Omron Sysmac Studio project ExamplePseudoUAMethod (Sysmac Studio 1.63.0.7, StandardProject)

# Controller Example: NX102-9000 version 1.64
Task PrimaryTask (priority 4, period or condition 4000): Methods, Math

VAR_GLOBAL
    Scalar_Static_Int32 : DINT;  (* network output *)
    Scalar_Static_Float : REAL;  (* network output *)
    Scalar_Static_String : STRING[64];  (* network output *)
END_VAR

PROGRAM Methods
VAR
    MyAdd : MtdMyAdd;
    MyMath : ClsMath;
END_VAR
IF P_First_Run THEN
	MyAdd.Execute := FALSE;
	MyMath.Enable := TRUE;
END_IF;

MyAdd();
MyMath();
END_PROGRAM

PROGRAM Math
VAR
    MyAdd : MtdMyAdd;
END_VAR
IF P_First_Run THEN
	MyAdd.Execute := FALSE;
END_IF;

MyAdd();
END_PROGRAM

FUNCTION_BLOCK MtdMyAdd
VAR_INPUT
    Execute : BOOL;
    In1 : UINT;
    In2 : UINT;
END_VAR
VAR_OUTPUT
    Out : UINT;
    Done : BOOL;
END_VAR
IF NOT Execute THEN
	Done := FALSE;
	
	RETURN;
END_IF;

IF Execute AND NOT Done THEN
	Out := In1 + In2;
	
	Done := TRUE;
END_IF;
END_FUNCTION_BLOCK

FUNCTION_BLOCK ClsMath
VAR
    MyAdd : MtdMyAdd;
END_VAR
VAR_INPUT
    Enable : BOOL;
END_VAR
VAR_OUTPUT
    Busy : BOOL;
END_VAR
IF Enable AND NOT Busy THEN
	Busy := TRUE;
ELSIF NOT Enable AND Busy THEN	
	MyAdd.Execute := FALSE;
	
	Busy := FALSE;
END_IF;

IF Busy THEN
	MyAdd();
END_IF;
END_FUNCTION_BLOCK